INTERFACE I_Sensor

PROPERTY PUBLIC isActive : BOOL
GET
END_GET
END_PROPERTY

PROPERTY PUBLIC isInactive : BOOL
GET
END_GET
END_PROPERTY

END_INTERFACE

(* stored: Version 1.1.0.1, ProductVersion 3.1.4024.12
   Itf I_Sensor: Id {b5c88b78-e437-49e5-95fc-4f9068651cbd}
   Property isActive: Id {e7245970-7437-4992-af4f-7275b0e63bc7}
   Get Get: Id {a9f3cd22-c8f4-4bf1-b2f1-86f98f841edb}
   Property isInactive: Id {afacba46-2b8b-442b-ba4a-1d0887f41add}
   Get Get: Id {4c1c4977-ca0b-40a5-b79f-c7ab0536be26} *)
